{attribute 'qualified_only'}
{attribute 'strict'}
TYPE RotationStates :
(
	Initialising,
	Start_Homing,
	Homing,
	Idle,
	Start_Move,
	Moving,
	Error
);
END_TYPE

(* stored: Version 1.1.0.1, ProductVersion 3.1.4024.11
   DUT RotationStates: Id {7d15cd09-b50d-481a-988b-32329a59abdf} *)
